// TIA Portal project "Two Axis Rotating lec 5" (V16)
// Vorlageprojekt für das Buch mit Zielsystem S7-1200

(* hardware
DEVICE "S7-1200-Station_1"  S7-1200 Station
   slot 0: "Baugruppenträger_0"  Rack  V1.0
   slot 1: "PLC_1"  CPU 1211C DC/DC/DC  6ES7 211-1AE40-0XB0  V4.1
*)

// ===== PLC "PLC_1"  CPU 1211C DC/DC/DC =====

VAR_GLOBAL   // PLC tag table "Standard-Variablentabelle"
   "Start Button" AT %I0.0 : Bool;
   "Stop Button" AT %I0.1 : Bool;
   "X Moving" AT %I0.5 : Bool;
   "Z Moving" AT %I0.6 : Bool;
   "Detected" AT %I0.7 : Bool;
   "Entry Conveyor" AT %Q0.0 : Bool;
   "Sorting Conveyor" AT %Q0.1 : Bool;
   "Small Conveyor" AT %Q0.2 : Bool;
   "Large Conveyor" AT %Q0.3 : Bool;
   "move X" AT %Q0.4 : Bool;
   "move Z" AT %Q0.5 : Bool;
   "Grab" AT %Q0.6 : Bool;
   "Rotate CW" AT %Q0.7 : Bool;
   "Rotate CCW" AT %Q1.0 : Bool;
   "Start Light" AT %Q1.1 : Bool;
   "Stop Light" AT %Q1.2 : Bool;
   "state0" AT %M0.1 : Bool;
   "state1" AT %M0.2 : Bool;
   "state2" AT %M0.3 : Bool;
   "state3" AT %M0.4 : Bool;
   "state4" AT %M0.5 : Bool;
   "state5" AT %M0.6 : Bool;
   "state6" AT %M0.7 : Bool;
   "state7" AT %M1.0 : Bool;
   "state8" AT %M1.1 : Bool;
   "state9" AT %M1.2 : Bool;
   "state10" AT %M1.3 : Bool;
   "state11" AT %M1.4 : Bool;
   "small BOX" AT %M4.0 : Bool;
   "large BOX" AT %M4.1 : Bool;
   "low sensor" AT %I0.2 : Bool;
   "high sensor" AT %I0.3 : Bool;
   "before TWO AXIS" AT %I0.4 : Bool;
   "Tag_1" AT %M8.0 : Bool;
   "Tag_2" AT %M8.1 : Bool;
   "Tag_3" AT %M8.3 : Bool;
   "rotating Detected" AT %I1.0 : Bool;
   "Tag_4" AT %M8.4 : Bool;
   "Tag_5" AT %M8.5 : Bool;
   "state12" AT %M1.5 : Bool;
   "state13" AT %M1.6 : Bool;
   "state14" AT %M1.7 : Bool;
   "state15" AT %M2.0 : Bool;
   "state16" AT %M2.1 : Bool;
   "state17" AT %M2.2 : Bool;
   "state18" AT %M2.3 : Bool;
   "state19" AT %M2.4 : Bool;
   "state20" AT %M2.5 : Bool;
   "state21" AT %M2.6 : Bool;
   "state22" AT %M2.7 : Bool;
   "state23" AT %M3.0 : Bool;
   "state24" AT %M3.1 : Bool;
   "state25" AT %M3.2 : Bool;
   "state26" AT %M3.3 : Bool;
   "Tag_6" AT %M8.6 : Bool;
   "Tag_7" AT %M9.0 : Bool;
   "Tag_8" AT %M9.1 : Bool;
   "Tag_9" AT %M9.2 : Bool;
   "Tag_10" AT %M9.3 : Bool;
   "Tag_11" AT %M9.4 : Bool;
   "Tag_12" AT %M9.5 : Bool;
END_VAR

FUNCTION "Cases" : Void   // FC1, LAD
{ S7_Optimized_Access := 'TRUE' }
VERSION : 0.1
   VAR_TEMP   // added for the SCL form of the ladder/FBD networks
      _w1 : Bool;
   END_VAR
BEGIN

REGION Network 1
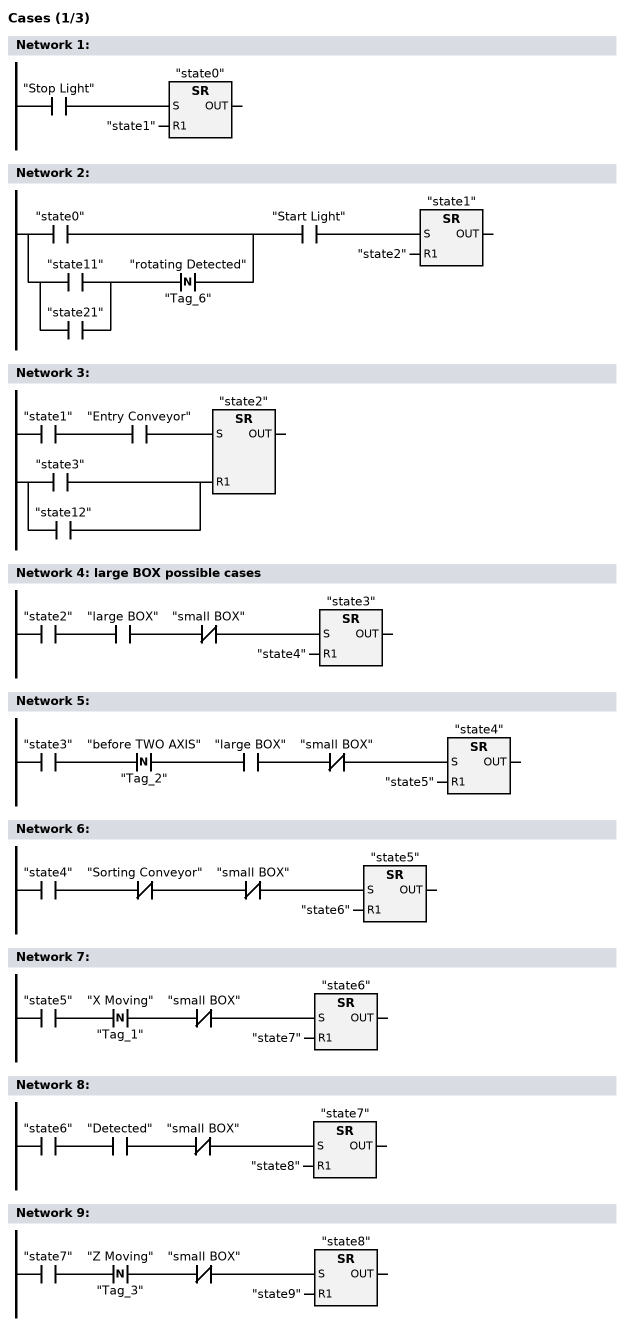
   RUNG wire#powerrail
      Contact( "Stop Light" )
      S_SR(operand := "state0", r1 := "state1")
   END_RUNG
   // the same network as SCL:
   IF "Stop Light" THEN
       "state0" := TRUE;   // SR flip-flop
   END_IF;
   IF "state1" THEN "state0" := FALSE; END_IF;
END_REGION

REGION Network 2
   RUNG wire#powerrail
      Contact( "state0" )
      wire#w1
      Contact( "Start Light" )
      S_SR(operand := "state1", r1 := "state2")
   END_RUNG
   RUNG wire#powerrail
      Contact( "state11" )
      wire#w2
      N_Contact(operand := "rotating Detected", bit := "Tag_6")
   END_RUNG wire#w1
   RUNG wire#powerrail
      Contact( "state21" )
   END_RUNG wire#w2
   // the same network as SCL:
   #_w1 := ("state11" OR "state21") AND NOT "rotating Detected" AND "Tag_6";   // falling edge of "rotating Detected"
   "Tag_6" := "rotating Detected";
   IF ("state0" OR #_w1) AND "Start Light" THEN
       "state1" := TRUE;   // SR flip-flop
   END_IF;
   IF "state2" THEN "state1" := FALSE; END_IF;
END_REGION

REGION Network 3
   RUNG wire#powerrail
      Contact( "state1" )
      Contact( "Entry Conveyor" )
      S_SR(operand := "state2", r1 := wire#w1)
   END_RUNG
   RUNG wire#powerrail
      Contact( "state3" )
   END_RUNG wire#w1
   RUNG wire#powerrail
      Contact( "state12" )
   END_RUNG wire#w1
   // the same network as SCL:
   IF "state1" AND "Entry Conveyor" THEN
       "state2" := TRUE;   // SR flip-flop
   END_IF;
   IF "state3" OR "state12" THEN "state2" := FALSE; END_IF;
END_REGION

REGION Network 4: large BOX possible cases
   RUNG wire#powerrail
      Contact( "state2" )
      Contact( "large BOX" )
      I_Contact( "small BOX" )
      S_SR(operand := "state3", r1 := "state4")
   END_RUNG
   // the same network as SCL:
   IF "state2" AND "large BOX" AND NOT "small BOX" THEN
       "state3" := TRUE;   // SR flip-flop
   END_IF;
   IF "state4" THEN "state3" := FALSE; END_IF;
END_REGION

REGION Network 5
   RUNG wire#powerrail
      Contact( "state3" )
      N_Contact(operand := "before TWO AXIS", bit := "Tag_2")
      Contact( "large BOX" )
      I_Contact( "small BOX" )
      S_SR(operand := "state4", r1 := "state5")
   END_RUNG
   // the same network as SCL:
   #_w1 := "state3" AND NOT "before TWO AXIS" AND "Tag_2";   // falling edge of "before TWO AXIS"
   "Tag_2" := "before TWO AXIS";
   IF #_w1 AND "large BOX" AND NOT "small BOX" THEN
       "state4" := TRUE;   // SR flip-flop
   END_IF;
   IF "state5" THEN "state4" := FALSE; END_IF;
END_REGION

REGION Network 6
   RUNG wire#powerrail
      Contact( "state4" )
      I_Contact( "Sorting Conveyor" )
      I_Contact( "small BOX" )
      S_SR(operand := "state5", r1 := "state6")
   END_RUNG
   // the same network as SCL:
   IF "state4" AND NOT "Sorting Conveyor" AND NOT "small BOX" THEN
       "state5" := TRUE;   // SR flip-flop
   END_IF;
   IF "state6" THEN "state5" := FALSE; END_IF;
END_REGION

REGION Network 7
   RUNG wire#powerrail
      Contact( "state5" )
      N_Contact(operand := "X Moving", bit := "Tag_1")
      I_Contact( "small BOX" )
      S_SR(operand := "state6", r1 := "state7")
   END_RUNG
   // the same network as SCL:
   #_w1 := "state5" AND NOT "X Moving" AND "Tag_1";   // falling edge of "X Moving"
   "Tag_1" := "X Moving";
   IF #_w1 AND NOT "small BOX" THEN
       "state6" := TRUE;   // SR flip-flop
   END_IF;
   IF "state7" THEN "state6" := FALSE; END_IF;
END_REGION

REGION Network 8
   RUNG wire#powerrail
      Contact( "state6" )
      Contact( "Detected" )
      I_Contact( "small BOX" )
      S_SR(operand := "state7", r1 := "state8")
   END_RUNG
   // the same network as SCL:
   IF "state6" AND "Detected" AND NOT "small BOX" THEN
       "state7" := TRUE;   // SR flip-flop
   END_IF;
   IF "state8" THEN "state7" := FALSE; END_IF;
END_REGION

REGION Network 9
   RUNG wire#powerrail
      Contact( "state7" )
      N_Contact(operand := "Z Moving", bit := "Tag_3")
      I_Contact( "small BOX" )
      S_SR(operand := "state8", r1 := "state9")
   END_RUNG
   // the same network as SCL:
   #_w1 := "state7" AND NOT "Z Moving" AND "Tag_3";   // falling edge of "Z Moving"
   "Tag_3" := "Z Moving";
   IF #_w1 AND NOT "small BOX" THEN
       "state8" := TRUE;   // SR flip-flop
   END_IF;
   IF "state9" THEN "state8" := FALSE; END_IF;
END_REGION

REGION Network 10
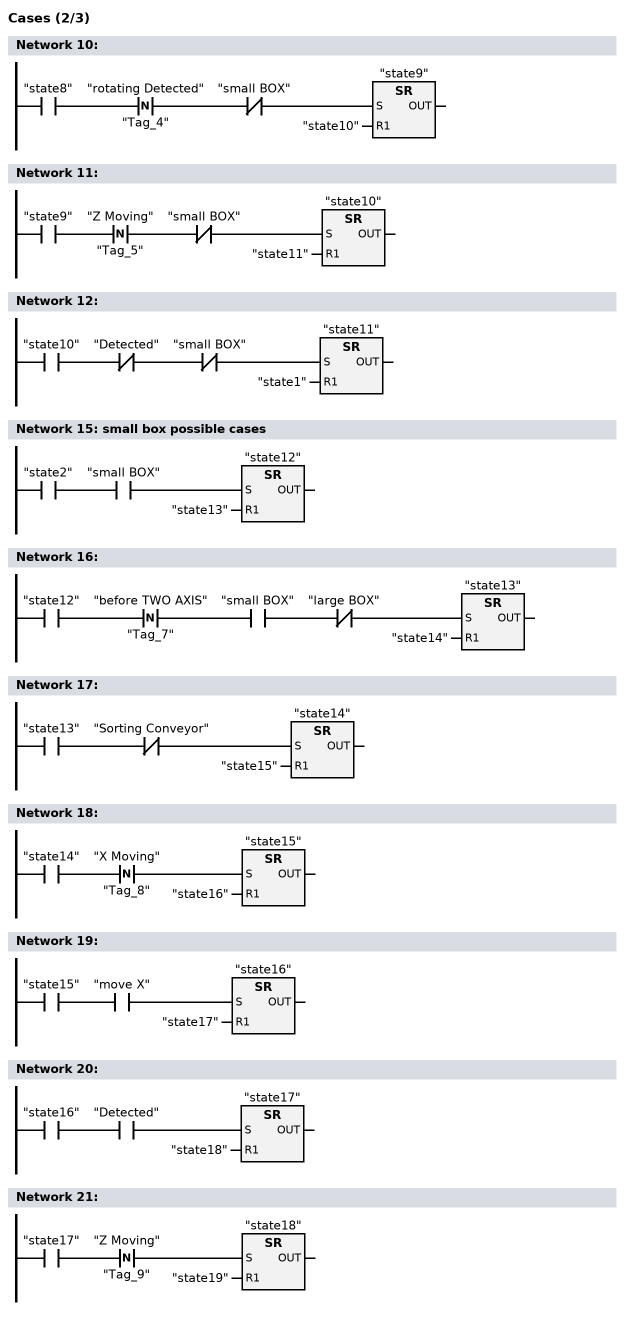
   RUNG wire#powerrail
      Contact( "state8" )
      N_Contact(operand := "rotating Detected", bit := "Tag_4")
      I_Contact( "small BOX" )
      S_SR(operand := "state9", r1 := "state10")
   END_RUNG
   // the same network as SCL:
   #_w1 := "state8" AND NOT "rotating Detected" AND "Tag_4";   // falling edge of "rotating Detected"
   "Tag_4" := "rotating Detected";
   IF #_w1 AND NOT "small BOX" THEN
       "state9" := TRUE;   // SR flip-flop
   END_IF;
   IF "state10" THEN "state9" := FALSE; END_IF;
END_REGION

REGION Network 11
   RUNG wire#powerrail
      Contact( "state9" )
      N_Contact(operand := "Z Moving", bit := "Tag_5")
      I_Contact( "small BOX" )
      S_SR(operand := "state10", r1 := "state11")
   END_RUNG
   // the same network as SCL:
   #_w1 := "state9" AND NOT "Z Moving" AND "Tag_5";   // falling edge of "Z Moving"
   "Tag_5" := "Z Moving";
   IF #_w1 AND NOT "small BOX" THEN
       "state10" := TRUE;   // SR flip-flop
   END_IF;
   IF "state11" THEN "state10" := FALSE; END_IF;
END_REGION

REGION Network 12
   RUNG wire#powerrail
      Contact( "state10" )
      I_Contact( "Detected" )
      I_Contact( "small BOX" )
      S_SR(operand := "state11", r1 := "state1")
   END_RUNG
   // the same network as SCL:
   IF "state10" AND NOT "Detected" AND NOT "small BOX" THEN
       "state11" := TRUE;   // SR flip-flop
   END_IF;
   IF "state1" THEN "state11" := FALSE; END_IF;
END_REGION

REGION Network 15: small box possible cases
   RUNG wire#powerrail
      Contact( "state2" )
      Contact( "small BOX" )
      S_SR(operand := "state12", r1 := "state13")
   END_RUNG
   // the same network as SCL:
   IF "state2" AND "small BOX" THEN
       "state12" := TRUE;   // SR flip-flop
   END_IF;
   IF "state13" THEN "state12" := FALSE; END_IF;
END_REGION

REGION Network 16
   RUNG wire#powerrail
      Contact( "state12" )
      N_Contact(operand := "before TWO AXIS", bit := "Tag_7")
      Contact( "small BOX" )
      I_Contact( "large BOX" )
      S_SR(operand := "state13", r1 := "state14")
   END_RUNG
   // the same network as SCL:
   #_w1 := "state12" AND NOT "before TWO AXIS" AND "Tag_7";   // falling edge of "before TWO AXIS"
   "Tag_7" := "before TWO AXIS";
   IF #_w1 AND "small BOX" AND NOT "large BOX" THEN
       "state13" := TRUE;   // SR flip-flop
   END_IF;
   IF "state14" THEN "state13" := FALSE; END_IF;
END_REGION

REGION Network 17
   RUNG wire#powerrail
      Contact( "state13" )
      I_Contact( "Sorting Conveyor" )
      S_SR(operand := "state14", r1 := "state15")
   END_RUNG
   // the same network as SCL:
   IF "state13" AND NOT "Sorting Conveyor" THEN
       "state14" := TRUE;   // SR flip-flop
   END_IF;
   IF "state15" THEN "state14" := FALSE; END_IF;
END_REGION

REGION Network 18
   RUNG wire#powerrail
      Contact( "state14" )
      N_Contact(operand := "X Moving", bit := "Tag_8")
      S_SR(operand := "state15", r1 := "state16")
   END_RUNG
   // the same network as SCL:
   #_w1 := "state14" AND NOT "X Moving" AND "Tag_8";   // falling edge of "X Moving"
   "Tag_8" := "X Moving";
   IF #_w1 THEN
       "state15" := TRUE;   // SR flip-flop
   END_IF;
   IF "state16" THEN "state15" := FALSE; END_IF;
END_REGION

REGION Network 19
   RUNG wire#powerrail
      Contact( "state15" )
      Contact( "move X" )
      S_SR(operand := "state16", r1 := "state17")
   END_RUNG
   // the same network as SCL:
   IF "state15" AND "move X" THEN
       "state16" := TRUE;   // SR flip-flop
   END_IF;
   IF "state17" THEN "state16" := FALSE; END_IF;
END_REGION

REGION Network 20
   RUNG wire#powerrail
      Contact( "state16" )
      Contact( "Detected" )
      S_SR(operand := "state17", r1 := "state18")
   END_RUNG
   // the same network as SCL:
   IF "state16" AND "Detected" THEN
       "state17" := TRUE;   // SR flip-flop
   END_IF;
   IF "state18" THEN "state17" := FALSE; END_IF;
END_REGION

REGION Network 21
   RUNG wire#powerrail
      Contact( "state17" )
      N_Contact(operand := "Z Moving", bit := "Tag_9")
      S_SR(operand := "state18", r1 := "state19")
   END_RUNG
   // the same network as SCL:
   #_w1 := "state17" AND NOT "Z Moving" AND "Tag_9";   // falling edge of "Z Moving"
   "Tag_9" := "Z Moving";
   IF #_w1 THEN
       "state18" := TRUE;   // SR flip-flop
   END_IF;
   IF "state19" THEN "state18" := FALSE; END_IF;
END_REGION

REGION Network 22
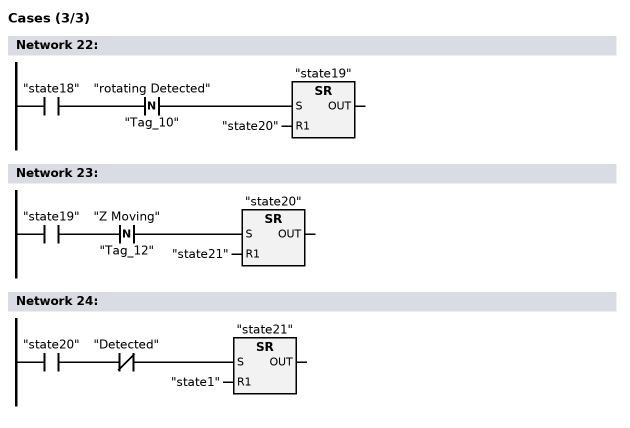
   RUNG wire#powerrail
      Contact( "state18" )
      N_Contact(operand := "rotating Detected", bit := "Tag_10")
      S_SR(operand := "state19", r1 := "state20")
   END_RUNG
   // the same network as SCL:
   #_w1 := "state18" AND NOT "rotating Detected" AND "Tag_10";   // falling edge of "rotating Detected"
   "Tag_10" := "rotating Detected";
   IF #_w1 THEN
       "state19" := TRUE;   // SR flip-flop
   END_IF;
   IF "state20" THEN "state19" := FALSE; END_IF;
END_REGION

REGION Network 23
   RUNG wire#powerrail
      Contact( "state19" )
      N_Contact(operand := "Z Moving", bit := "Tag_12")
      S_SR(operand := "state20", r1 := "state21")
   END_RUNG
   // the same network as SCL:
   #_w1 := "state19" AND NOT "Z Moving" AND "Tag_12";   // falling edge of "Z Moving"
   "Tag_12" := "Z Moving";
   IF #_w1 THEN
       "state20" := TRUE;   // SR flip-flop
   END_IF;
   IF "state21" THEN "state20" := FALSE; END_IF;
END_REGION

REGION Network 24
   RUNG wire#powerrail
      Contact( "state20" )
      I_Contact( "Detected" )
      S_SR(operand := "state21", r1 := "state1")
   END_RUNG
   // the same network as SCL:
   IF "state20" AND NOT "Detected" THEN
       "state21" := TRUE;   // SR flip-flop
   END_IF;
   IF "state1" THEN "state21" := FALSE; END_IF;
END_REGION
END_FUNCTION

FUNCTION "Outputs" : Void   // FC2, LAD
{ S7_Optimized_Access := 'TRUE' }
VERSION : 0.1
BEGIN

REGION Network 1
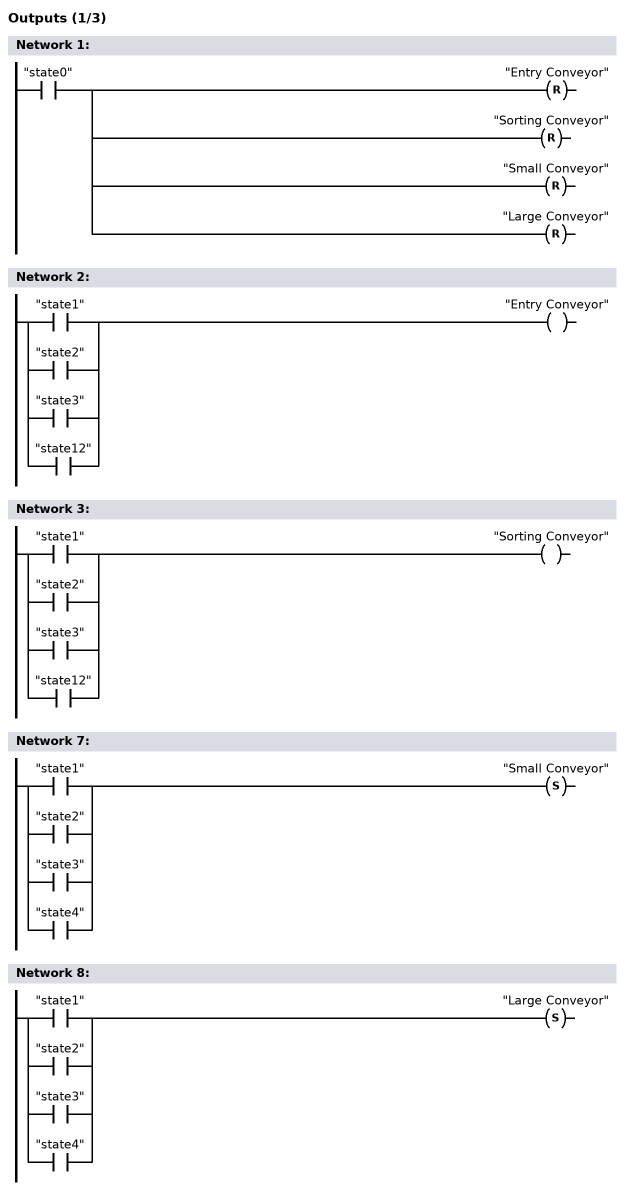
   RUNG wire#powerrail
      Contact( "state0" )
      wire#w1
      R_Coil( "Entry Conveyor" )
   END_RUNG
   RUNG wire#w1
      R_Coil( "Sorting Conveyor" )
   END_RUNG
   RUNG wire#w1
      R_Coil( "Small Conveyor" )
   END_RUNG
   RUNG wire#w1
      R_Coil( "Large Conveyor" )
   END_RUNG
   // the same network as SCL:
   IF "state0" THEN
       "Entry Conveyor" := FALSE;
       "Sorting Conveyor" := FALSE;
       "Small Conveyor" := FALSE;
       "Large Conveyor" := FALSE;
   END_IF;
END_REGION

REGION Network 2
   RUNG wire#powerrail
      Contact( "state1" )
      wire#w1
      Coil( "Entry Conveyor" )
   END_RUNG
   RUNG wire#powerrail
      Contact( "state2" )
   END_RUNG wire#w1
   RUNG wire#powerrail
      Contact( "state3" )
   END_RUNG wire#w1
   RUNG wire#powerrail
      Contact( "state12" )
   END_RUNG wire#w1
   // the same network as SCL:
   "Entry Conveyor" := "state1" OR "state2" OR "state3" OR "state12";
END_REGION

REGION Network 3
   RUNG wire#powerrail
      Contact( "state1" )
      wire#w1
      Coil( "Sorting Conveyor" )
   END_RUNG
   RUNG wire#powerrail
      Contact( "state2" )
   END_RUNG wire#w1
   RUNG wire#powerrail
      Contact( "state3" )
   END_RUNG wire#w1
   RUNG wire#powerrail
      Contact( "state12" )
   END_RUNG wire#w1
   // the same network as SCL:
   "Sorting Conveyor" := "state1" OR "state2" OR "state3" OR "state12";
END_REGION

REGION Network 7
   RUNG wire#powerrail
      Contact( "state1" )
      wire#w1
      S_Coil( "Small Conveyor" )
   END_RUNG
   RUNG wire#powerrail
      Contact( "state2" )
   END_RUNG wire#w1
   RUNG wire#powerrail
      Contact( "state3" )
   END_RUNG wire#w1
   RUNG wire#powerrail
      Contact( "state4" )
   END_RUNG wire#w1
   // the same network as SCL:
   IF "state1" OR "state2" OR "state3" OR "state4" THEN "Small Conveyor" := TRUE; END_IF;
END_REGION

REGION Network 8
   RUNG wire#powerrail
      Contact( "state1" )
      wire#w1
      S_Coil( "Large Conveyor" )
   END_RUNG
   RUNG wire#powerrail
      Contact( "state2" )
   END_RUNG wire#w1
   RUNG wire#powerrail
      Contact( "state3" )
   END_RUNG wire#w1
   RUNG wire#powerrail
      Contact( "state4" )
   END_RUNG wire#w1
   // the same network as SCL:
   IF "state1" OR "state2" OR "state3" OR "state4" THEN "Large Conveyor" := TRUE; END_IF;
END_REGION

REGION Network 9
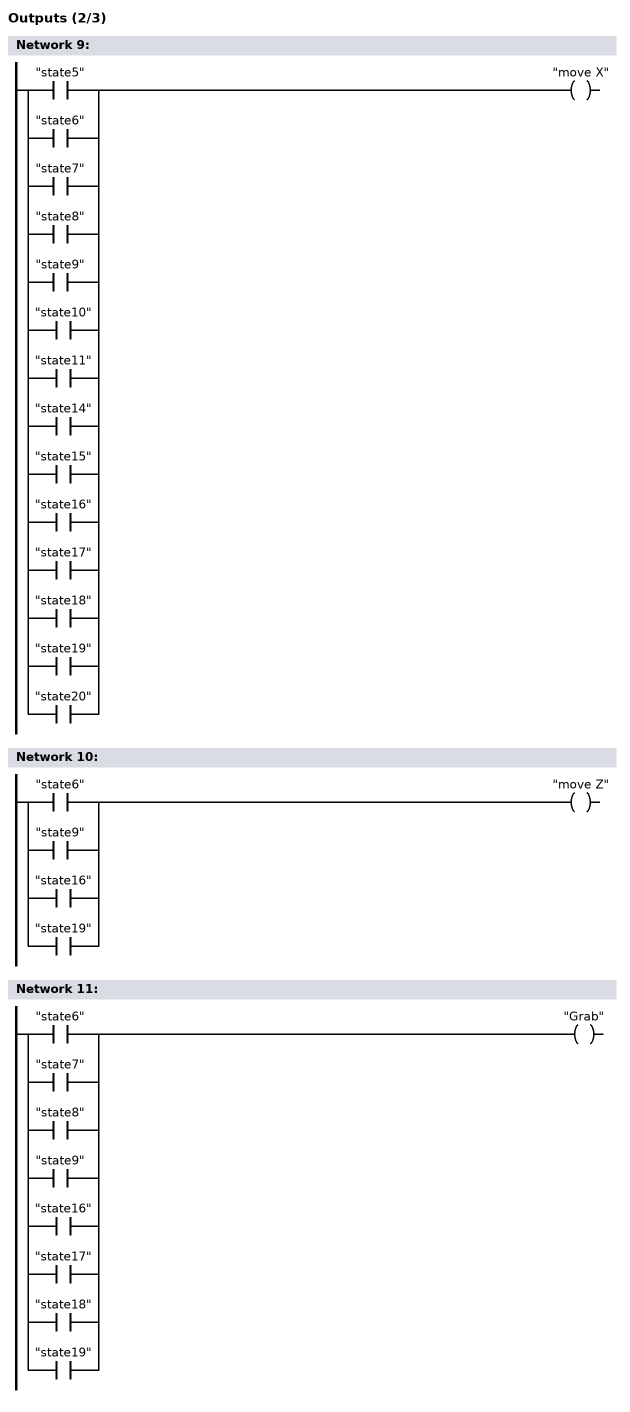
   RUNG wire#powerrail
      Contact( "state5" )
      wire#w1
      Coil( "move X" )
   END_RUNG
   RUNG wire#powerrail
      Contact( "state6" )
   END_RUNG wire#w1
   RUNG wire#powerrail
      Contact( "state7" )
   END_RUNG wire#w1
   RUNG wire#powerrail
      Contact( "state8" )
   END_RUNG wire#w1
   RUNG wire#powerrail
      Contact( "state9" )
   END_RUNG wire#w1
   RUNG wire#powerrail
      Contact( "state10" )
   END_RUNG wire#w1
   RUNG wire#powerrail
      Contact( "state11" )
   END_RUNG wire#w1
   RUNG wire#powerrail
      Contact( "state14" )
   END_RUNG wire#w1
   RUNG wire#powerrail
      Contact( "state15" )
   END_RUNG wire#w1
   RUNG wire#powerrail
      Contact( "state16" )
   END_RUNG wire#w1
   RUNG wire#powerrail
      Contact( "state17" )
   END_RUNG wire#w1
   RUNG wire#powerrail
      Contact( "state18" )
   END_RUNG wire#w1
   RUNG wire#powerrail
      Contact( "state19" )
   END_RUNG wire#w1
   RUNG wire#powerrail
      Contact( "state20" )
   END_RUNG wire#w1
   // the same network as SCL:
   "move X" := "state5" OR "state6" OR "state7" OR "state8" OR "state9" OR "state10" OR "state11" OR "state14" OR "state15" OR "state16" OR "state17" OR "state18" OR "state19" OR "state20";
END_REGION

REGION Network 10
   RUNG wire#powerrail
      Contact( "state6" )
      wire#w1
      Coil( "move Z" )
   END_RUNG
   RUNG wire#powerrail
      Contact( "state9" )
   END_RUNG wire#w1
   RUNG wire#powerrail
      Contact( "state16" )
   END_RUNG wire#w1
   RUNG wire#powerrail
      Contact( "state19" )
   END_RUNG wire#w1
   // the same network as SCL:
   "move Z" := "state6" OR "state9" OR "state16" OR "state19";
END_REGION

REGION Network 11
   RUNG wire#powerrail
      Contact( "state6" )
      wire#w1
      Coil( "Grab" )
   END_RUNG
   RUNG wire#powerrail
      Contact( "state7" )
   END_RUNG wire#w1
   RUNG wire#powerrail
      Contact( "state8" )
   END_RUNG wire#w1
   RUNG wire#powerrail
      Contact( "state9" )
   END_RUNG wire#w1
   RUNG wire#powerrail
      Contact( "state16" )
   END_RUNG wire#w1
   RUNG wire#powerrail
      Contact( "state17" )
   END_RUNG wire#w1
   RUNG wire#powerrail
      Contact( "state18" )
   END_RUNG wire#w1
   RUNG wire#powerrail
      Contact( "state19" )
   END_RUNG wire#w1
   // the same network as SCL:
   "Grab" := "state6" OR "state7" OR "state8" OR "state9" OR "state16" OR "state17" OR "state18" OR "state19";
END_REGION

REGION Network 12
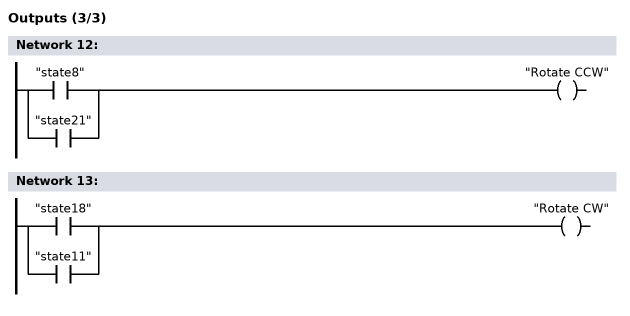
   RUNG wire#powerrail
      Contact( "state8" )
      wire#w1
      Coil( "Rotate CCW" )
   END_RUNG
   RUNG wire#powerrail
      Contact( "state21" )
   END_RUNG wire#w1
   // the same network as SCL:
   "Rotate CCW" := "state8" OR "state21";
END_REGION

REGION Network 13
   RUNG wire#powerrail
      Contact( "state18" )
      wire#w1
      Coil( "Rotate CW" )
   END_RUNG
   RUNG wire#powerrail
      Contact( "state11" )
   END_RUNG wire#w1
   // the same network as SCL:
   "Rotate CW" := "state18" OR "state11";
END_REGION
END_FUNCTION

FUNCTION "start stop" : Void   // FC3, LAD
{ S7_Optimized_Access := 'TRUE' }
VERSION : 0.1
BEGIN

REGION Network 1
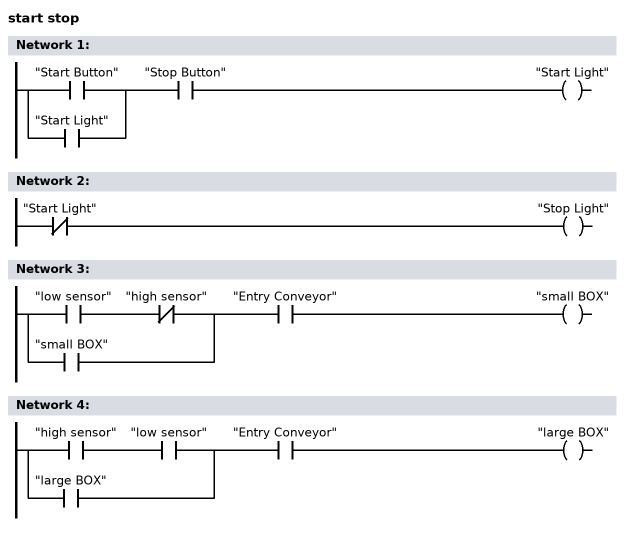
   RUNG wire#powerrail
      Contact( "Start Button" )
      wire#w1
      Contact( "Stop Button" )
      Coil( "Start Light" )
   END_RUNG
   RUNG wire#powerrail
      Contact( "Start Light" )
   END_RUNG wire#w1
   // the same network as SCL:
   "Start Light" := ("Start Button" OR "Start Light") AND "Stop Button";
END_REGION

REGION Network 2
   RUNG wire#powerrail
      I_Contact( "Start Light" )
      Coil( "Stop Light" )
   END_RUNG
   // the same network as SCL:
   "Stop Light" := NOT "Start Light";
END_REGION

REGION Network 3
   RUNG wire#powerrail
      Contact( "low sensor" )
      I_Contact( "high sensor" )
      wire#w1
      Contact( "Entry Conveyor" )
      Coil( "small BOX" )
   END_RUNG
   RUNG wire#powerrail
      Contact( "small BOX" )
   END_RUNG wire#w1
   // the same network as SCL:
   "small BOX" := (("low sensor" AND NOT "high sensor") OR "small BOX") AND "Entry Conveyor";
END_REGION

REGION Network 4
   RUNG wire#powerrail
      Contact( "high sensor" )
      Contact( "low sensor" )
      wire#w1
      Contact( "Entry Conveyor" )
      Coil( "large BOX" )
   END_RUNG
   RUNG wire#powerrail
      Contact( "large BOX" )
   END_RUNG wire#w1
   // the same network as SCL:
   "large BOX" := (("high sensor" AND "low sensor") OR "large BOX") AND "Entry Conveyor";
END_REGION
END_FUNCTION

FUNCTION "MHJ-PLC-Lab-Function-S71200" : Void   // FC9000, SCL
{ S7_Optimized_Access := 'TRUE' }
VERSION : 0.1
   VAR_TEMP
      rdTimeReturn : Int;
      outputTime : DTL;
      SyncVal : Byte;
      forVal : Int;
      forVal_2 : Int;
      Value : Byte;
   END_VAR
   VAR CONSTANT
      CompVal : Byte := 16#34;
      Value_01 : Byte := 16#11;
      Value_01_DW : DWord := 16#A165_D992;
      Value_02_DW : DWord := 16#58BE_4401;
   END_VAR
BEGIN

   #Value:=PEEK(area := 16#82,
        dbNumber := 0,
        byteOffset := 511);
   #Value := #Value + 1;

   POKE(area := 16#82,
        dbNumber := 0,
        byteOffset := 511,
        value := #Value);

   POKE(area:=16#81,
        dbNumber:=0,
        byteOffset:=1016,
        value:=#Value_01_DW);
   POKE(area := 16#81,
        dbNumber := 0,
        byteOffset := 1020,
        value := #Value_02_DW);

   POKE(area := 16#81,
        dbNumber := 0,
        byteOffset := 511,
        value := B#16#00);

   FOR #forVal := 0 TO 120 DO
       FOR #forVal_2:=0 TO 10 DO
           #rdTimeReturn:=RD_SYS_T(#outputTime);
           #rdTimeReturn := WR_SYS_T(#outputTime);
           #rdTimeReturn := RD_SYS_T(#outputTime);
           #rdTimeReturn := WR_SYS_T(#outputTime);
       END_FOR;
       #SyncVal:= PEEK(area := 16#81,
                      dbNumber := 0,
                      byteOffset := 511);
       IF #SyncVal = #CompVal THEN
          GOTO M_1;
       END_IF;
   END_FOR;
   RETURN;

   M_1:
   POKE(area := 16#81,
        dbNumber := 0,
        byteOffset := 511,
        value := B#16#0);
END_FUNCTION

ORGANIZATION_BLOCK "Main"   // OB1, LAD, ProgramCycle
TITLE = "Main Program Sweep (Cycle)"
{ S7_Optimized_Access := 'TRUE' }
VERSION : 0.1
   VAR_INPUT
      Initial_Call : Bool;   // Initial call of this OB
      Remanence : Bool;   // =True, if remanent data are available
   END_VAR
BEGIN

REGION Network 1: Konnektierungsbaustein für PLC-Lab
   // Im Netzwerk 1 wird der Konnektierungsbaustein für PLC-Lab aufgerufen.
   // Dieser Aufruf darf nicht entfernt werden!
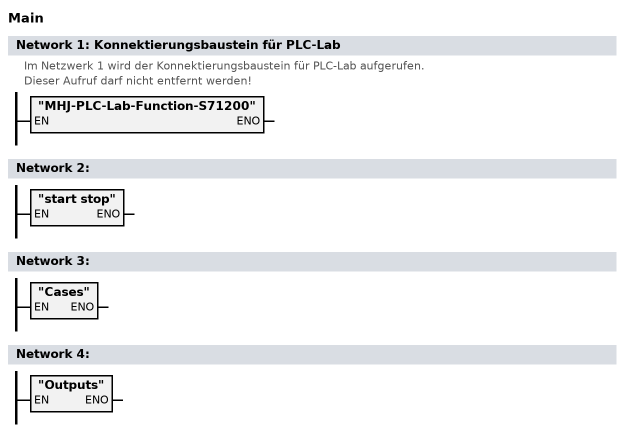
   RUNG wire#powerrail
      "MHJ-PLC-Lab-Function-S71200"()
   END_RUNG
   // the same network as SCL:
   "MHJ-PLC-Lab-Function-S71200"();
END_REGION

REGION Network 2
   RUNG wire#powerrail
      "start stop"()
   END_RUNG
   // the same network as SCL:
   "start stop"();
END_REGION

REGION Network 3
   RUNG wire#powerrail
      "Cases"()
   END_RUNG
   // the same network as SCL:
   "Cases"();
END_REGION

REGION Network 4
   RUNG wire#powerrail
      "Outputs"()
   END_RUNG
   // the same network as SCL:
   "Outputs"();
END_REGION
END_ORGANIZATION_BLOCK

ORGANIZATION_BLOCK "Startup"   // OB100, LAD, Startup
TITLE = "Complete Restart"
{ S7_Optimized_Access := 'TRUE' }
VERSION : 0.1
   VAR_INPUT
      LostRetentive : Bool;   // True if retentive data are lost
      LostRTC : Bool;   // True if date and time are lost
   END_VAR
BEGIN

REGION Network 1
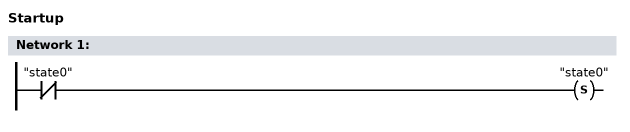
   RUNG wire#powerrail
      I_Contact( "state0" )
      S_Coil( "state0" )
   END_RUNG
   // the same network as SCL:
   IF NOT "state0" THEN "state0" := TRUE; END_IF;
END_REGION
END_ORGANIZATION_BLOCK